FUNCTION_BLOCK SectionDelivery
  (* Standard: 61499-2 *)
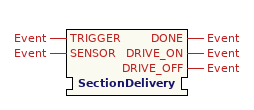
  EVENT_INPUT
    TRIGGER;
    SENSOR;
  END_EVENT
  EVENT_OUTPUT
    DONE;
    DRIVE_ON;
    DRIVE_OFF;
  END_EVENT
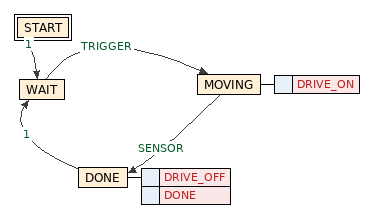
  EC_STATES
    START;
    MOVING : -> DRIVE_ON;
    WAIT;
    DONE : -> DRIVE_OFF, -> DONE;
  END_STATES
  EC_TRANSITIONS
    START TO WAIT := 1;
    WAIT TO MOVING := TRIGGER;
    MOVING TO DONE := SENSOR;
    DONE TO WAIT := 1;
  END_TRANSITIONS
  ALGORITHM INIT IN ST:

  END_ALGORITHM
  ALGORITHM REQ IN ST:

  END_ALGORITHM
END_FUNCTION_BLOCK
